// TIA Portal V16 export
// export: Created 2022-04-14T22:38:37.872773Z, ExportSetting WithDefaults, DisplayName Totally Integrated Automation Portal, DisplayVersion V16, DisplayName TIA Portal Version Control Interface, DisplayVersion V16, DisplayName TIA Portal Openness, DisplayVersion V16, DisplayName STEP 7 Professional, DisplayVersion V16, DisplayName STEP 7 Safety, DisplayVersion V16, DisplayName WinCC Professional, DisplayVersion V16
FUNCTION_BLOCK "05 Pusher"   // FB3, LAD
{ S7_Optimized_Access := 'TRUE' }
VERSION : 0.1
// stored: AutoNumber true, IsIECCheckEnabled false, IsRetainMemResEnabled false, MemoryReserve 100, SetENOAutomatically false, UDAEnableTagReadback false
   VAR_TEMP   // added for the SCL form of the ladder/FBD networks
      _w1 : Bool;
      _w2 : Bool;
   END_VAR
BEGIN

REGION Network 1: Sorting by height 1
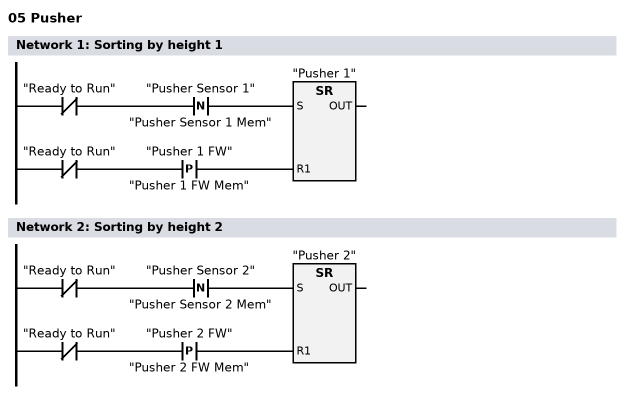
   RUNG wire#powerrail
      I_Contact( "Ready to Run" )
      N_Contact(operand := "Pusher Sensor 1", bit := "Pusher Sensor 1 Mem")
      S_SR(operand := "Pusher 1", r1 := wire#w1)
   END_RUNG
   RUNG wire#powerrail
      I_Contact( "Ready to Run" )
      P_Contact(operand := "Pusher 1 FW", bit := "Pusher 1 FW Mem")
   END_RUNG wire#w1
   // the same network as SCL:
   #_w1 := NOT "Ready to Run" AND NOT "Pusher Sensor 1" AND "Pusher Sensor 1 Mem";   // falling edge of "Pusher Sensor 1"
   "Pusher Sensor 1 Mem" := "Pusher Sensor 1";
   #_w2 := NOT "Ready to Run" AND "Pusher 1 FW" AND NOT "Pusher 1 FW Mem";   // rising edge of "Pusher 1 FW"
   "Pusher 1 FW Mem" := "Pusher 1 FW";
   IF #_w1 THEN
       "Pusher 1" := TRUE;   // SR flip-flop
   END_IF;
   IF #_w2 THEN "Pusher 1" := FALSE; END_IF;
END_REGION

REGION Network 2: Sorting by height 2
   RUNG wire#powerrail
      I_Contact( "Ready to Run" )
      N_Contact(operand := "Pusher Sensor 2", bit := "Pusher Sensor 2 Mem")
      S_SR(operand := "Pusher 2", r1 := wire#w1)
   END_RUNG
   RUNG wire#powerrail
      I_Contact( "Ready to Run" )
      P_Contact(operand := "Pusher 2 FW", bit := "Pusher 2 FW Mem")
   END_RUNG wire#w1
   // the same network as SCL:
   #_w1 := NOT "Ready to Run" AND NOT "Pusher Sensor 2" AND "Pusher Sensor 2 Mem";   // falling edge of "Pusher Sensor 2"
   "Pusher Sensor 2 Mem" := "Pusher Sensor 2";
   #_w2 := NOT "Ready to Run" AND "Pusher 2 FW" AND NOT "Pusher 2 FW Mem";   // rising edge of "Pusher 2 FW"
   "Pusher 2 FW Mem" := "Pusher 2 FW";
   IF #_w1 THEN
       "Pusher 2" := TRUE;   // SR flip-flop
   END_IF;
   IF #_w2 THEN "Pusher 2" := FALSE; END_IF;
END_REGION
END_FUNCTION_BLOCK
